FUNCTION_BLOCK EL72x1_DMC
VAR_INPUT
END_VAR
VAR_OUTPUT
END_VAR
VAR
	//Properties
	_acceleration : UINT := 4000; 	//default to 4s accel
	_deceleration : UINT := 4000;	//default to 4s decel
	_startType : UINT := 1; 		//default to abs moves
	_scale : REAL := 360; 			//default to 360 degree scale factor
	
	//Locals
	dmc_inputs AT%I* : DMC_Ins;
	dmc_outputs AT%q* : DMC_Outs;
	xMove: BOOL;
	iMove: INT;
	
	posDemand : REAL;
	currentPos : REAL;
END_VAR

MoveSequence();

dmc_outputs.DMC_DrvOuts.TargetPosition := REAL_TO_UDINT(posDemand * (1048576/360));
currentPos := UDINT_TO_REAL( dmc_inputs.DMC_Inputs.ActualPosition)*(360.0/1048576.0);

PROPERTY PUBLIC Acceleration : uint
GET
Acceleration := _acceleration;
END_GET
SET
_acceleration := Acceleration;
END_SET
END_PROPERTY

PROPERTY PUBLIC Deceleration : uint
GET
Deceleration := _deceleration;
END_GET
SET
_deceleration := Deceleration;
END_SET
END_PROPERTY

METHOD PUBLIC Enable : BOOL
VAR_INPUT
END_VAR
IF dmc_inputs.DMC_Drv_Status.ReadyToEnable THEN
	dmc_outputs.DMC_Drv_Ctrl.Enable := TRUE;
END_IF
END_METHOD

PROPERTY PUBLIC Enabled : bool
GET
Enabled := dmc_inputs.DMC_Drv_Status.Ready AND dmc_inputs.DMC_POS_Status.ReadyToExecute;
END_GET
END_PROPERTY

PROPERTY PUBLIC Error : bool
GET
Error := dmc_inputs.DMC_Drv_Status.Error;
END_GET
END_PROPERTY

METHOD PUBLIC MoveAxis : BOOL
VAR_INPUT
	PositioningControl : real;
	Velocity : INT;
END_VAR
dmc_outputs.DMC_DrvOuts.TargetPosition := REAL_TO_UDINT(PositioningControl*(1048576/_scale));
dmc_outputs.DMC_DrvOuts.TargetVelocity := Velocity;
dmc_outputs.DMC_DrvOuts.StartType := _startType;
dmc_outputs.DMC_DrvOuts.TargetAcceleration := _acceleration;
dmc_outputs.DMC_DrvOuts.TargetDeceleration := _deceleration;
xMove := TRUE;
MoveAxis := TRUE;
END_METHOD

METHOD PRIVATE MoveSequence : BOOL
VAR_INPUT
END_VAR
CASE iMove OF 
	0: 
		IF dmc_inputs.DMC_POS_Status.ReadyToExecute AND xMove THEN
			xMove := FALSE;
			iMove := 10;
		END_IF
	10:
		dmc_outputs.DMC_POS_Ctrl.Execute := TRUE;
		IF dmc_inputs.DMC_POS_Status.Busy THEN
			iMove := 20;
		END_IF
	20:
		IF NOT dmc_inputs.DMC_POS_Status.Busy THEN
			IF dmc_inputs.DMC_POS_Status.InTarget THEN
				iMove := 0;
			ELSE
				iMove :=99;
			END_IF
			dmc_outputs.DMC_POS_Ctrl.Execute := FALSE;
		END_IF
END_CASE
END_METHOD

PROPERTY PUBLIC Scale : real
GET
Scale := _scale;
END_GET
SET
_scale := Scale;
END_SET
END_PROPERTY

PROPERTY PUBLIC StartType : uint
GET
StartType := _startType;
END_GET
SET
_startType := StartType;
END_SET
END_PROPERTY

END_FUNCTION_BLOCK

(* stored: Version 1.1.0.1, ProductVersion 3.1.4024.9
   POU EL72x1_DMC: Id {5d7a0ba8-888d-479f-99c5-25bd7d6d845a}, SpecialFunc None
   Property Acceleration: Id {0f489025-7d66-4b39-8820-723a22fd0dc7}
   Get Get: Id {8d8d8e4e-1dd6-42ed-965b-623973f9ecb6}
   Set Set: Id {10052c2f-e003-4a0a-9fbc-e4a0bcc611ca}
   Property Deceleration: Id {4c65d767-dd9c-4b66-8970-767316944559}
   Get Get: Id {08331d35-7b36-4dec-8f1c-7df4ae7b9476}
   Set Set: Id {e313fc1e-0f34-408c-8d2a-98f5fb58defb}
   Method Enable: Id {3e7b7545-0028-4626-8ed8-9f5042b5ff68}
   Property Enabled: Id {e8331ba0-e7ef-4ea0-b2e5-be04bf4e43f1}
   Get Get: Id {c719c9f7-93a2-43d8-a292-341fc754ab8b}
   Property Error: Id {5b09fc6d-ff5b-47fe-a5cb-3a624411a0d5}
   Get Get: Id {272c0756-e2fe-4fc8-876b-a614711307f4}
   Method MoveAxis: Id {e4fb2b63-faf3-42a6-9470-f798dcffe77f}
   Method MoveSequence: Id {35f8abeb-e88f-43b1-8480-fa08e614a561}
   Property Scale: Id {e75115b2-c129-4232-a701-3301b1398b5d}
   Get Get: Id {698f0f1c-a8e7-4bed-9992-4fa56eeb8d19}
   Set Set: Id {c8f37d03-d4a0-44de-9559-bed6432fa9f3}
   Property StartType: Id {7e2cf6ed-c7f3-4a23-bfb6-dbb9aa440449}
   Get Get: Id {5fb5db65-0608-4b42-ab84-bd34f014a280}
   Set Set: Id {1d2f504a-5036-487e-a5ea-4229b3174833} *)
